% RSLogix 500 project HOA_BAK001.RSS, saved by version 8.30.00.16 %
PROJECT "HOA"    % processor: Bul.1763 MicroLogix 1100 Series B %

PROGRAM FILES
  LAD 2 "MAIN"  3 rungs
  LAD 3 "DIG IO"  5 rungs
  LAD 4 "CONTROLS"  1 rungs

DATA FILES
  O0 OUTPUT  5 elements
  I1 INPUT  7 elements
  S2 STATUS  66 elements
  B3 BINARY  1 elements
  T4 TIMER  1 elements
  C5 COUNTER  1 elements
  R6 CONTROL  1 elements
  N7 INTEGER  1 elements
  F8 FLOAT  1 elements

LADDER 2 "MAIN"
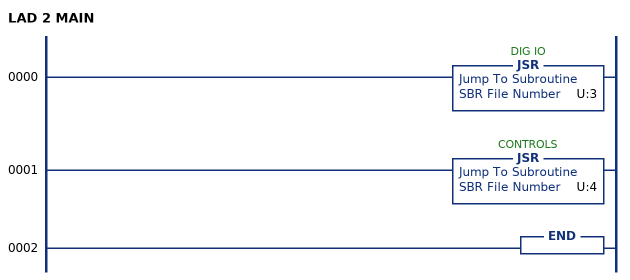
% Rung: 0 %  % edit flag set %
SOR JSR U:3 EOR
%   U:3  "DIG IO" %
% Rung: 1 %  % edit flag set %
SOR JSR U:4 EOR
%   U:4  "CONTROLS" %
% Rung: 2 %
SOR END EOR

LADDER 3 "DIG IO"
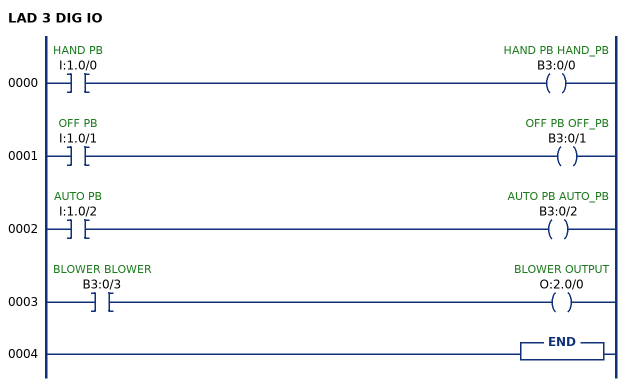
% Rung: 0 %  % edit flag set %
SOR XIC I:1.0/0 OTE B3:0/0 EOR
%   I:1.0/0  "HAND PB" %
%   B3:0/0  HAND_PB  "HAND PB" %
% Rung: 1 %  % edit flag set %
SOR XIC I:1.0/1 OTE B3:0/1 EOR
%   I:1.0/1  "OFF PB" %
%   B3:0/1  OFF_PB  "OFF PB" %
% Rung: 2 %  % edit flag set %
SOR XIC I:1.0/2 OTE B3:0/2 EOR
%   I:1.0/2  "AUTO PB" %
%   B3:0/2  AUTO_PB  "AUTO PB" %
% Rung: 3 %  % edit flag set %
SOR XIC B3:0/3 OTE O:2.0/0 EOR
%   B3:0/3  BLOWER  "BLOWER" %
%   O:2.0/0  "BLOWER OUTPUT" %
% Rung: 4 %
SOR END EOR

REVISION NOTES
  0: ADDED DIG IO
